FUNCTION_BLOCK Test_TStreamAdd_Read_STRING EXTENDS TUnitTestBase
VAR
    Stream : TStream(StreamLength := 2);
    TestString : STRING := '111111111 222222222 333333333 444444444 555555555 666666666 777777777 888888888 ';
END_VAR



Stream.Init(2);

Stream.Add_STRING(TestString);
    
Assertion.AssertEquals_UDINT(
    Expected := 81,
    Actual := Stream.Position,
    VariableName := 'Stream.Position');
    
Stream.Seek(0);

Assertion.AssertEquals_STRING(
    Expected := TestString,
    Actual := Stream.Read_STRING(),
    VariableName := 'Stream.Read_STRING()');
    
Assertion.AssertEquals_UDINT(
    Expected := 81,
    Actual := Stream.Position,
    VariableName := 'Stream.Position');
    
    
TestFinished();

END_FUNCTION_BLOCK

(* stored: Version 1.1.0.1, ProductVersion 3.1.4024.4
   POU Test_TStreamAdd_Read_STRING: Id {ab5097ac-b326-40f7-a5ee-e13d182a186b}, SpecialFunc None *)
